TYPE ST_Configuration :
STRUCT
	/// debug logging configuration
	stLogConfig			: ST_LoggingConfig;
	
	stVar2FileConfig	: ST_Var2File_Config;
END_STRUCT
END_TYPE

(* stored: Version 1.1.0.1
   DUT ST_Configuration: Id {c9977f54-26d6-4eaf-871b-6a2f2409e879} *)
